(* IEC 61131-3 sources: json/test, 18 files *)

(* ---- CompareArray.st ---- *)
NAMESPACE Simatic.Ax.Json
    FUNCTION CompareArray : BOOL
        VAR_INPUT
            first : ARRAY[*] OF CHAR;
            scnd : ARRAY[*] OF CHAR;
            count : INT;
        END_VAR
        VAR_TEMP
            i : DINT;
            sFirst : DINT;
            sScnd : DINT;
            eFirst : DINT;
            eScnd : DINT;
            res : BOOL;
            _count : DINT;
        END_VAR

        sFirst := LOWER_BOUND(first, 1);
        sScnd := LOWER_BOUND(scnd, 1);
        eFirst := UPPER_BOUND(first, 1);
        eScnd := UPPER_BOUND(scnd, 1);

        _count := count;

        IF ((eFirst - sFirst + 1) < count) THEN
            CompareArray := FALSE;
            RETURN;
        END_IF;
        IF ((eScnd - sScnd + 1) < count) THEN
            CompareArray := FALSE;
            RETURN;
        END_IF;

        IF _count > (eFirst - sFirst + 1) THEN
            _count := eFirst - sFirst + 1;
        END_IF;

        FOR i := 0 TO _count - 1 DO
            res := first[i + sFirst] = scnd[i + sScnd];
            IF (res = FALSE) THEN
                CompareArray := FALSE;
                RETURN;
            END_IF;
        END_FOR;
        CompareArray := TRUE;
    END_FUNCTION
END_NAMESPACE

(* ---- FindKeyInBuffer.st ---- *)
USING Simatic.Ax.Conversion;
USING AxUnit.Assert;
USING System.Strings;
using Simatic.Ax.Json;

NAMESPACE Deserializer

{TestFixture}
CLASS Test_FindKeyInBuffer
    VAR protected
        doc : JsonDocument;
        testString : STRING := 'works!';
        buffer : ARRAY[1..999] OF CHAR;
    END_VAR

    METHOD PUBLIC ConvertStringToCharArray
        VAR_INPUT
            inputstring: string;
        end_var
        VAR_TEMP
            stringLength : int;
            index : Int;
        end_var

        stringLength := LengthOf(inputstring);

        FOR Index := 1 TO stringlength DO
            buffer[index] := inputstring[index];
        END_FOR;

    END_METHOD

    {Test}
    METHOD PUBLIC Test_ConvertStringToCharArray
            THIS.ConvertStringToCharArray(testString);
            Equal('w', buffer[1]);
            Equal('o', buffer[2]);
            Equal('r', buffer[3]);
            Equal('k', buffer[4]);
            Equal('s', buffer[5]);
            Equal('!', buffer[6]);
    END_METHOD

END_CLASS

{Test}
FUNCTION GetACharInString
    VAR_TEMP
        e : STRING := 'hallo';
        c : CHAR;
    end_var
        c := e[1];
        Equal(c, 'h');
END_FUNCTION

END_NAMESPACE

(* ---- StringAssert.st ---- *)
USING AxUnit.ResultFunctions;
USING System.Strings;

NAMESPACE AxUnit.Assert
    FUNCTION PUBLIC Equal
        VAR_INPUT
            actual : String;
            expected: String;
            {CallerFilePath}
            file : WSTRING[1024];
            {CallerLineNumber}
            line : INT;
        END_VAR

        IF actual = expected THEN
            axunit_Succeed();
        ELSE
            axunit_Fail(Concat('Expected ', ', but found '), file, line);
        END_IF;

    END_FUNCTION
END_NAMESPACE

(* ---- test.st ---- *)
USING AxUnit.Assert;

NAMESPACE Simatic.Ax.Json
    FUNCTION test : Int
        VAR_INPUT

        END_VAR
        test := 3;
    END_FUNCTION

    {TestFixture}
    CLASS MyTestFixture
        {Test}
        METHOD PUBLIC function_returns_alwasy_4
            Equal(expected := 4, actual := test());
            ; // AxUnit.Assert.Equal(y, x)
        END_METHOD
    END_CLASS

END_NAMESPACE

(* ---- TestFindKeyInBuffer.st ---- *)
USING Simatic.Ax.Conversion;
USING AxUnit.Assert;
USING System.Strings;
using Simatic.Ax.Json;

NAMESPACE Deserializer

{TestFixture}
CLASS Test_FindKeyInBuffer
    VAR protected
        doc : JsonDocument;
        key: STRING := 'key';
        testString : STRING := 'works!';
        buffer : ARRAY[0..999] OF CHAR;
    END_VAR

    {Test}
    Method Public Test_FindAKeyPosition_in_JSON_OneEntry
        VAR
            JSON_Entry: STRING := '{"Key1": "Element1"}';

            len:DINT;
            keyStart : int;
            keyEnd : int;
            keysFound: int;
        END_VAR

        len:= Strings.ToArray(str := JSON_Entry, arr := doc.buffer);

        keysFound := doc.FindKey(keyStart, keyEnd);

        //index is 0 based, not 1 based!
        Equal(2, keyStart);
        Equal(5, keyEnd);
        Equal(keysFound, 1);
    END_Method

    {Test}
    Method Public Test_FindKeysPosition_in_JSON_2Entries
        VAR
            JSON_Entry: STRING := '{"Key1": "Element1","Key2": 1234}';

            len:DINT;
            keyStart : int;
            keyEnd : int;
            keysFound: int;
        END_VAR

        len:= Strings.ToArray(str := JSON_Entry, arr := doc.buffer);

        keysFound := doc.FindKey(keyStart, keyEnd);

        //index is 0 based, not 1 based!
        Equal(21, keyStart);
        Equal(24, keyEnd);
        Equal(keysFound, 2);
    END_Method

    {Test}
    Method Public Test_KeyIsInIndexSpan_FindsKey
        VAR
            len:DINT;
            keyStart : int := 0;
            keyEnd : int := 2;
            keyFound: BOOL;

            test: bool := true;
        END_VAR

        len:= Strings.ToArray(str := key, arr := doc.buffer);

        keyFound := doc.KeyIsInIndexSpan(REF(key), keyStart, keyEnd);
        Equal(TRUE, keyFound);

        key := 'not';
        keyFound := doc.KeyIsInIndexSpan(REF(key), keyStart, keyEnd);
        Equal(FALSE, keyFound);
    END_Method

    //start with FindKey, in a string, Get Back Key and value. Make TryParse out of it (provide key). Nachteil: json wird jedes mal durchsucht. Test: Stringlänge! (Refto string?)

END_CLASS

{Test}
FUNCTION GetACharInString
    VAR_TEMP
        e : STRING := 'hallo';
        c : CHAR;
    end_var
        c := e[1];
        Equal(c, 'h');
END_FUNCTION

END_NAMESPACE

(* ---- Example.st ---- *)
USING Simatic.Ax.Json;
USING AxUnit.Assert;

NAMESPACE Simatic.Ax
    CLASS JsonExample
        VAR PUBLIC

        END_VAR
        VAR PROTECTED
            doc : JsonDocument;
            e1 : JsonDInt := (Key := 'Element1', Value := 1);
            e2 : JsonDInt := (Key := 'Element2', Value := 2);
            e3 : JsonDInt := (Key := 'Element3', Value := 3);
            o1 : JsonObject := (Key := 'NestedObject');

        END_VAR

        METHOD PUBLIC Init;
            // Example String:
            // {"Element1": 1, {"Element2": 2, "Element3": 3}}
            doc.AddElement(e1);
            doc.AddElement(o1);
            o1.AddElement(e2);
            o1.AddElement(e3);
        END_METHOD

        METHOD PUBLIC ToString : STRING
            ToString := doc.ToString();
        END_METHOD
    END_CLASS
END_NAMESPACE

NAMESPACE Simatic.Ax
    {TestFixture}
    CLASS TestExample
        VAR PROTECTED
            _ex : JsonExample;
        END_VAR

        {Test}
        METHOD PUBLIC TestExample_and_check_returned_string
            VAR_TEMP
                _expStr : STRING;
                _actStr : STRING;
            END_VAR
            _ex.Init();
            _expStr := '{"Element1": 1, "NestedObject": {"Element2": 2, "Element3": 3}}';
            _actStr := _ex.ToString();
            Equal(expected := _actStr, actual := _expStr);
        END_METHOD
    END_CLASS

END_NAMESPACE

(* ---- ItemTest.st ---- *)
USING AxUnit.Assert;
USING System.Strings;

NAMESPACE Simatic.Ax.Json
    {TestFixture}
    CLASS TestJsonElementsDint

        VAR PROTECTED
            e : Properties.DoubleInt := (value := 999, key := 'test');
        END_VAR

        {Test}
        METHOD PUBLIC Test_Tostring_with_999_expect_test_999
            Equal(expected := e.ToString(), actual := '"test": "999"');
        END_METHOD

        {Test}
        METHOD PUBLIC Test_Tostring_with_Minus_999_expect_test_Minus_999
            Equal(expected := e.ToString(), actual := '"test": "999"');
        END_METHOD

    END_CLASS
END_NAMESPACE

(* ---- ItemTestDint.st ---- *)
USING AxUnit.Assert;
USING System.Strings;

NAMESPACE Simatic.Ax.Json
    {TestFixture}
    CLASS TestJsonElementsDint

        VAR PROTECTED
            e : JsonDoubleInt := (value := 999, key := 'test');
            e2 : JsonDoubleInt := (value := -999, key := 'second_key');
        END_VAR

        {Test}
        METHOD PUBLIC Test_Tostring_with_999_expect_test_999
            VAR_TEMP
                _str : STRING;
            END_VAR
            _str := e.ToString();
            Equal(expected := _str, actual := '"test": 999');
        END_METHOD

        {Test}
        METHOD PUBLIC Test_Tostring_with_Minus_999_expect_test_Minus_999
            Equal(expected := e2.ToString(), actual := '"second_key": -999');
        END_METHOD

    END_CLASS
END_NAMESPACE

(* ---- ItemTestInt.st ---- *)
USING AxUnit.Assert;
USING System.Strings;
USING Simatic.Ax.Conversion;

NAMESPACE Simatic.Ax.Json
    {TestFixture}
    CLASS TestJsonElementsInt

        VAR PROTECTED
            e : JsonInt := (value := 999, key := 'test');
            e2 : JsonInt := (value := -999, key := 'second_key');
            s_test_999 : STRING := '"test": 999';
            s_test_minus_999 : STRING := '"second_key": -999';
            cmpBuff : ARRAY[0..20] OF CHAR;
            doc : JsonDocument;
        END_VAR

        {Test}
        METHOD PUBLIC Test_Tostring_with_999_expect_test_999
            VAR_TEMP
                _str : STRING;
            END_VAR
            _str := e.ToString();
            Equal(expected := _str, actual := s_test_999);
        END_METHOD

        {Test}
        METHOD PUBLIC Test_Tostring_with_Minus_999_expect_test_Minus_999
            Equal(expected := e2.ToString(), actual := s_test_minus_999);
        END_METHOD

        {Test}
        METHOD PUBLIC TestSerialize_s_test_999
            VAR_TEMP
                len : DINT;
                res : BOOL;
            END_VAR
            e.Serialize(REF(doc));

            len := Strings.ToArray(str := s_test_999, arr := cmpBuff);
            res := CompareArray(first := doc.buffer, scnd := cmpBuff, count := TO_INT(len));
            Equal(expected := TRUE, actual := res);

        END_METHOD

        {Test}
        METHOD PUBLIC TestSerialize_s_test_minus_999
            VAR_TEMP
                len : DINT;
                res : BOOL;
            END_VAR

            e2.Serialize(REF(doc));
            len := Strings.ToArray(str := s_test_minus_999, arr := cmpBuff);
            res := CompareArray(first := doc.buffer, scnd := cmpBuff, count := TO_INT(len));
            Equal(expected := TRUE, actual := res);

        END_METHOD
    END_CLASS
END_NAMESPACE

(* ---- ItemTestLint.st ---- *)
USING AxUnit.Assert;
USING System.Strings;

NAMESPACE Simatic.Ax.Json
    {TestFixture}
    CLASS TestJsonElementsLint

        VAR PROTECTED
            e : JsonLInt := (Value := 999, Key := 'test');
            e2 : JsonLInt := (Value := -999, Key := 'second_key');
        END_VAR

        {Test}
        METHOD PUBLIC Test_Tostring_with_999_expect_test_999
            VAR_TEMP
                _str : STRING;
            END_VAR
            _str := e.ToString();
            Equal(expected := _str, actual := '"test": 999');
        END_METHOD

        {Test}
        METHOD PUBLIC Test_Tostring_with_Minus_999_expect_test_Minus_999
            Equal(expected := e2.ToString(), actual := '"second_key": -999');
        END_METHOD

    END_CLASS
END_NAMESPACE

(* ---- ItemTestSint.st ---- *)
USING AxUnit.Assert;
USING System.Strings;
USING Simatic.Ax.Conversion;

NAMESPACE Simatic.Ax.Json
    {TestFixture}
    CLASS TestJsonElementsSInt

        VAR PROTECTED
            e : JsonSInt := (Value := SINT#127, Key := 'test');
            e2 : JsonSInt := (Value := SINT#-128, Key := 'second_key');
            s_test_127 : STRING := '"test": 127';
            s_test_minus_128 : STRING := '"second_key": -128';
            cmpBuff : ARRAY[0..20] OF CHAR;
            doc : JsonDocument;
        END_VAR

        {Test}
        METHOD PUBLIC Test_Tostring_with_999_expect_test_999
            VAR_TEMP
                _str : STRING;
            END_VAR
            _str := e.ToString();
            Equal(expected := _str, actual := s_test_127);
        END_METHOD

        {Test}
        METHOD PUBLIC Test_Tostring_with_Minus_999_expect_test_Minus_999
            Equal(expected := e2.ToString(), actual := s_test_minus_128);
        END_METHOD

        {Test}
        METHOD PUBLIC TestSerialize_s_test_999
            VAR_TEMP
                len : DINT;
                res : BOOL;
            END_VAR
            e.Serialize(REF(doc));

            len := Strings.ToArray(str := s_test_127, arr := cmpBuff);
            res := CompareArray(first := doc.buffer, scnd := cmpBuff, count := TO_INT(len));
            Equal(expected := TRUE, actual := res);

        END_METHOD

        {Test}
        METHOD PUBLIC TestSerialize_s_test_minus_999
            VAR_TEMP
                len : DINT;
                res : BOOL;
            END_VAR

            e2.Serialize(REF(doc));
            len := Strings.ToArray(str := s_test_minus_128, arr := cmpBuff);
            res := CompareArray(first := doc.buffer, scnd := cmpBuff, count := TO_INT(len));
            Equal(expected := TRUE, actual := res);

        END_METHOD
    END_CLASS
END_NAMESPACE

(* ---- ItemTestUSint.st ---- *)
USING AxUnit.Assert;
USING System.Strings;
USING Simatic.Ax.Conversion;

NAMESPACE Simatic.Ax.Json
    {TestFixture}
    CLASS TestJsonElementsUSInt

        VAR PROTECTED
            e : JsonUSInt := (Value := USINT#255, Key := 'test');
            e2 : JsonUSInt := (Value := USINT#0, Key := 'second_key');
            s_test_max : STRING := '"test": 255';
            s_test_minus_min : STRING := '"second_key": 0';
            cmpBuff : ARRAY[0..20] OF CHAR;
            doc : JsonDocument;
        END_VAR

        {Test}
        METHOD PUBLIC Test_Tostring_with_999_expect_test_999
            VAR_TEMP
                _str : STRING;
            END_VAR
            _str := e.ToString();
            Equal(expected := _str, actual := s_test_max);
        END_METHOD

        {Test}
        METHOD PUBLIC Test_Tostring_with_Minus_999_expect_test_Minus_999
            Equal(expected := e2.ToString(), actual := s_test_minus_min);
        END_METHOD

        {Test}
        METHOD PUBLIC TestSerialize_s_test_999
            VAR_TEMP
                len : DINT;
                res : BOOL;
            END_VAR
            e.Serialize(REF(doc));

            len := Strings.ToArray(str := s_test_max, arr := cmpBuff);
            res := CompareArray(first := doc.buffer, scnd := cmpBuff, count := TO_INT(len));
            Equal(expected := TRUE, actual := res);

        END_METHOD

        {Test}
        METHOD PUBLIC TestSerialize_s_test_minus_999
            VAR_TEMP
                len : DINT;
                res : BOOL;
            END_VAR

            e2.Serialize(REF(doc));
            len := Strings.ToArray(str := s_test_minus_min, arr := cmpBuff);
            res := CompareArray(first := doc.buffer, scnd := cmpBuff, count := TO_INT(len));
            Equal(expected := TRUE, actual := res);

        END_METHOD
    END_CLASS
END_NAMESPACE

(* ---- TestCompareArray.st ---- *)
USING AxUnit.Assert;
USING System.Strings;

NAMESPACE Simatic.Ax.Json
    {TestFixture}
    CLASS TestCompareArrayOfChar
        VAR
            a0_4_abcde : ARRAY[0..4] OF CHAR := ['a', 'b', 'c', 'd', 'e'];
            a0_4_abcdf : ARRAY[0..4] OF CHAR := ['a', 'b', 'c', 'd', 'f'];
            a0_4_12345 : ARRAY[0..4] OF CHAR := ['1', '2', '3', '4', '5'];
            a2_6_abcde : ARRAY[2..6] OF CHAR := ['a', 'b', 'c', 'd', 'e'];
            a2_6_12345 : ARRAY[2..6] OF CHAR := ['1', '2', '3', '4', '5'];
            a0_2_abc : ARRAY[0..2] OF CHAR := ['a', 'b', 'c'];
        END_VAR

        {Test}
        METHOD PUBLIC Copare_same_ArrayWithLengt5_Expect_TRUE
            VAR_TEMP
                res : BOOL;
            END_VAR
            res := CompareArray(a0_4_abcde, a0_4_abcde, 5);
            Equal(expected := TRUE, actual := res);

            res := CompareArray(a2_6_abcde, a2_6_abcde, 5);
            Equal(expected := TRUE, actual := res);
        END_METHOD

        {Test}
        METHOD PUBLIC Copare_different_ArrayWithLengt5_Expect_FALSE
            VAR_TEMP
                res : BOOL;
            END_VAR
            res := CompareArray(a0_4_abcde, a2_6_12345, 5);
            Equal(expected := FALSE, actual := res);

            res := CompareArray(a2_6_abcde, a0_4_12345, 5);
            Equal(expected := FALSE, actual := res);

            res := CompareArray(a0_4_abcde, a0_4_abcdf, 5);
            Equal(expected := FALSE, actual := res);

        END_METHOD

        {Test}
        METHOD PUBLIC Copare_different_ArrayWithLengt4_Expect_TRUE
            VAR_TEMP
                res : BOOL;
            END_VAR

            res := CompareArray(a0_4_abcde, a0_4_abcdf, 4);
            Equal(expected := TRUE, actual := res);

        END_METHOD

        {Test}
        METHOD PUBLIC Copare_same_ArrayWithLengt4_Expect_TRUE
            VAR_TEMP
                res : BOOL;
            END_VAR
            res := CompareArray(a0_4_abcde, a0_4_abcde, 4);
            Equal(expected := TRUE, actual := res);

            res := CompareArray(a2_6_abcde, a2_6_abcde, 4);
            Equal(expected := TRUE, actual := res);
        END_METHOD

        {Test}
        METHOD PUBLIC Copare_mixed_indices_ArrayWithLengt5_Expect_TRUE
            VAR_TEMP
                res : BOOL;
            END_VAR
            res := CompareArray(a0_4_abcde, a2_6_abcde, 5);
            Equal(expected := TRUE, actual := res);
        END_METHOD

        {Test}
        METHOD PUBLIC Copare_different_ArrayWithLengt4_Expect_FALSE
            VAR_TEMP
                res : BOOL;
            END_VAR
            res := CompareArray(a0_4_abcde, a2_6_12345, 4);
            Equal(expected := FALSE, actual := res);

            res := CompareArray(a2_6_abcde, a0_4_12345, 4);
            Equal(expected := FALSE, actual := res);
        END_METHOD

        {Test}
        METHOD PUBLIC Copare_different_lenght_ArrayWithLengt5_and_3_Expect_TRUE
            VAR_TEMP
                res : BOOL;
            END_VAR
            res := CompareArray(a0_4_abcde, a0_2_abc, 2);
            Equal(expected := TRUE, actual := res);

            res := CompareArray(a0_2_abc, a0_4_abcde, 2);
            Equal(expected := TRUE, actual := res);

            res := CompareArray(a0_4_abcde, a0_2_abc, 3);
            Equal(expected := TRUE, actual := res);

            res := CompareArray(a0_2_abc, a0_4_abcde, 3);
            Equal(expected := TRUE, actual := res);

            res := CompareArray(a0_4_abcde, a0_2_abc, 4);
            Equal(expected := FALSE, actual := res);

            res := CompareArray(a0_2_abc, a0_4_abcde, 4);
            Equal(expected := FALSE, actual := res);

            res := CompareArray(a0_4_abcde, a0_2_abc, 5);
            Equal(expected := FALSE, actual := res);

            res := CompareArray(a0_2_abc, a0_4_abcde, 5);
            Equal(expected := FALSE, actual := res);

            res := CompareArray(a0_4_abcde, a0_2_abc, 6);
            Equal(expected := FALSE, actual := res);

            res := CompareArray(a0_2_abc, a0_4_abcde, 6);
            Equal(expected := FALSE, actual := res);

        END_METHOD

    END_CLASS
END_NAMESPACE

(* ---- TestDoubleNestetdObject.st ---- *)
USING AxUnit.Assert;
USING System.Strings;
USING Simatic.Ax.Conversion;

NAMESPACE Simatic.Ax.Json
    {TestFixture}
    CLASS TestDoubleNestetdObject

        VAR PROTECTED
            e1 : JsonDInt := (Value := 999, Key := 'e1');
            o1 : JsonObject := (Key := 'O1');
            o2 : JsonObject := (Key := 'O2');
            o3 : JsonObject := (Key := 'O3');

            // {"O1": {"O2": "O3""e1" :}}
                                // 01234567890123456789012345678901234567890
            expString : STRING := '{"O1": {"O2": {"O3": {"e1": 999}}}}';

            actString : STRING;
            res : BOOL;
            doc : JsonDocument;
            cmpBuff : ARRAY[0..399] OF CHAR;
            len : DINT;
        END_VAR

        {Test}
        METHOD PUBLIC Test_Build_nested_object_And_expect_correct_JSON
            VAR_TEMP
                _to : IJsonElementMuteable;
                _elem : IJsonElement;
            END_VAR

            o3.AddElement(e1);
            o2.AddElement(o3);
            o1.AddElement(o2);
            doc.AddElement(o1);
            doc.Serialize(doc.buffer);

            len := Strings.ToArray(str := expString, arr := cmpBuff);
            res := CompareArray(first := doc.buffer, scnd := cmpBuff, count := TO_INT(len));
            Equal(expected := TRUE, actual := res);
        END_METHOD

    END_CLASS
END_NAMESPACE

(* ---- TestFindValueInBuffer.st ---- *)
USING Simatic.Ax.Conversion;
USING AxUnit.Assert;
USING System.Strings;
using Simatic.Ax.Json;

NAMESPACE Deserializer

{TestFixture}
CLASS Test_FindValueInBuffer
    VAR protected
        doc : JsonDocument;

        key: STRING;
        value: STRING;
        testIndex1: INT;
        testIndex2: INT;
    END_VAR

    {Test}
    Method Public Test_GetValueFromIndex_GetValue
        VAR
            len: DINT;
        END_VAR

        len:= Strings.ToArray(str := '1234', arr := doc.buffer);

        testIndex1:= 0; testIndex2 := 3;
        value:= doc.GetValueFromIndex(REF(testIndex1), REF(testIndex2));

        Equal('1234', value);

    END_Method

    {Test}
    Method Public Test_GetValueFromIndex_GetValue_withSpaces
        VAR
            len: DINT;
        END_VAR

        len:= Strings.ToArray(str := '    1234    ', arr := doc.buffer);

        testIndex1:= 0; testIndex2 := 10;
        value:= doc.GetValueFromIndex(REF(testIndex1), REF(testIndex2));

        Equal('1234', value);

    END_Method

    {Test}
    Method Public Test_GetValueFromIndex_GetValue_withQuotationMarks
        VAR
            len: DINT;
        END_VAR

        len:= Strings.ToArray(str := ' "1234"      ', arr := doc.buffer);

        testIndex1:= 0; testIndex2 := 10;
        value:= doc.GetValueFromIndex(REF(testIndex1), REF(testIndex2));

        Equal('1234', value);

    END_Method

END_CLASS

END_NAMESPACE

(* ---- TestJsonDocument.st ---- *)
USING AxUnit.Assert;
USING System.Strings;
USING Simatic.Ax.Conversion;

NAMESPACE Simatic.Ax.Json
    {TestFixture}
    CLASS TestJsonDocument

        VAR PROTECTED
            e : JsonDoubleInt := (value := 999, key := 'test');
            e2 : JsonDoubleInt := (value := -999, key := 'second_key');
            e3 : JsonDoubleInt := (value := 1, key := '3rd');
            doc : JsonDocument;
            o2 : JsonObject := (key := 'Name');

            iElem : IJsonElement;
            rElem : REF_TO JsonDoubleInt;
            expArray : ARRAY[0..399] OF CHAR;
            expArrayCnt : DINT;
            expString : STRING;
            actString : STRING;
            result : BOOL;

        END_VAR

        {Test}
        METHOD PUBLIC Test_Empty_object_ToString_Expect_empty_object

            // expected string
            expString := '{}';

            actString :=  doc.ToString();
            Equal(expected := expString, actual := actString);

            // Test Serialize
            expArrayCnt := Strings.ToArray(str := expString, arr := expArray);
            doc.Serialize(doc.buffer);
            result := CompareArray(first := doc.buffer, scnd := expArray, count := TO_INT(expArrayCnt));
            Equal(expected := TRUE, actual := result);

        END_METHOD

        {Test}
        METHOD PUBLIC Test_object_with_one_element_ToString_Expect_correct_string
            // expected string
            expString := '{"test": 999}';

            doc.AddElement(e);
            actString := doc.ToString();
            Equal(expected := expString, actual := actString);

            // Test Serialize
            expArrayCnt := Strings.ToArray(str := expString, arr := expArray);
            doc.Serialize(doc.buffer);
            result := CompareArray(first := doc.buffer, scnd := expArray, count := TO_INT(expArrayCnt));
            Equal(expected := TRUE, actual := result);
        END_METHOD

        {Test}
        METHOD PUBLIC Test_object_in_object_expect_nested_object
            // expected string
            expString := '{{}}';

            doc.AddElement(o2);
            Equal(expected := doc.ToString(), actual := expString);

            // Test Serialize
            expArrayCnt := Strings.ToArray(str := expString, arr := expArray);
            doc.Serialize(doc.buffer);
            result := CompareArray(first := doc.buffer, scnd := expArray, count := TO_INT(expArrayCnt));
            Equal(expected := TRUE, actual := result);
        END_METHOD

        {Test}
        METHOD PUBLIC Test_object_in_object_with_property_expect_nested_object
            // expected string
            expString := '{"Name": {"test": 999}}';

            doc.AddElement(o2);
            o2.AddElement(e);

            actString := doc.ToString();
            Equal(expected := actString, actual := expString);

            // Test Serialize
            expArrayCnt := Strings.ToArray(str := expString, arr := expArray);
            doc.Serialize(doc.buffer);
            result := CompareArray(first := doc.buffer, scnd := expArray, count := TO_INT(expArrayCnt));
            Equal(expected := TRUE, actual := result);
        END_METHOD

        {Test}
        METHOD PUBLIC Test_object_with_two_property_expect_object
            // expected string
            expString := '{"test": 999, "second_key": -999}';

            doc.AddElement(e);
            doc.AddElement(e2);
            Equal(expected := doc.ToString(), actual := expString);

            // Test Serialize
            expArrayCnt := Strings.ToArray(str := expString, arr := expArray);
            doc.Serialize(doc.buffer);
            result := CompareArray(first := doc.buffer, scnd := expArray, count := TO_INT(expArrayCnt));
            Equal(expected := TRUE, actual := result);
        END_METHOD

        {Test}
        METHOD PUBLIC Test_object_with_three_property_expect_object
            // expected string
            expString := '{"test": 999, "second_key": -999, "3rd": 1}';

            doc.AddElement(e);
            doc.AddElement(e2);
            doc.AddElement(e3);
            Equal(expected := doc.ToString(), actual := expString);

            // Test Serialize
            expArrayCnt := Strings.ToArray(str := expString, arr := expArray);
            doc.Serialize(doc.buffer);
            result := CompareArray(first := doc.buffer, scnd := expArray, count := TO_INT(expArrayCnt));
            Equal(expected := TRUE, actual := result);
        END_METHOD

        {Test}
        METHOD PUBLIC CreateTwoObjects_and_expect_correct_values
            // expected string
            expString := '{"test": 999, "second_key": -999}';

            doc.AddElement(e);
            doc.AddElement(e2);
            Equal(expected := doc.ToString(), actual := expString);

            // expected string
            expString := '"NestedObject": {"3rd": 1}';

            o2.key := 'NestedObject';
            o2.AddElement(e3);
            actString := o2.ToString();
            Equal(expected := expString, actual := actString);

            //            0        1         2         3         4         5         6         7
            //            1234567890123456789012345678901234567890123456789012345678901234567890
            expString := '{"test": 999, "second_key": -999, "NestedObject": {"3rd": 1}}';

            doc.AddElement(o2);
            actString := o2.ToString();

            actString := doc.ToString();
            Equal(expected := expString , actual := actString);

            // // Test Serialize
            // expArrayCnt := Strings.ToArray(str := expString, arr := expArray);
            // doc.Serialize(doc.buffer);
            // result := CompareArray(first := doc.buffer, scnd := expArray, count := TO_INT(expArrayCnt));
            // Equal(expected := TRUE, actual := result);
        END_METHOD
    END_CLASS
END_NAMESPACE

(* ---- TestJsonLongDocument.st ---- *)
USING AxUnit.Assert;
USING System.Strings;
USING Simatic.Ax.Conversion;
NAMESPACE Simatic.Ax.Json
    {TestFixture}
    CLASS TestJsonLongDocument

        VAR PROTECTED
            e1 : JsonInt := (Key := 'elem1', Value := 0);
            e2 : JsonLInt := (Key := 'elem2', Value := 1);
            e3 : JsonDInt := (Key := 'elem3', Value := 2);
            doc :JsonDocument;
        END_VAR

        METHOD PUBLIC MyMethod
            doc.AddElement(e1);
            doc.AddElement(e2);
            doc.AddElement(e3);
            doc.Serialize(doc.buffer); //--> {elem1: 0, elem2: 1, elem3: 2}\n
            // nice to have --> doc.Deserialize('{elem1: 99, elem2: 100, elem3: 111}\n')
        END_METHOD

    END_CLASS

END_NAMESPACE

(* ---- TestJsonObject.st ---- *)
USING AxUnit.Assert;
USING System.Strings;
USING Simatic.Ax.Conversion;

NAMESPACE Simatic.Ax.Json
    {TestFixture}
    CLASS TestJsonObject

        VAR PROTECTED
            e : JsonDoubleInt := (value := 999, key := 'test');
            e2 : JsonDoubleInt := (value := -999, key := 'second_key');
            e3 : JsonDoubleInt := (value := 1, key := '3rd');
            o : JsonObject := (key := 'Name');
            doc : JsonDocument;
            cmpBuff : ARRAY[0..399] OF CHAR;
            len : DINT;
        END_VAR

        {Test}
        METHOD PUBLIC Test_Empty_object_ToString_Expect_empty_object
            VAR_TEMP
                _expStr : STRING;
                _actStr : STRING;
            END_VAR

            // {}
            _expStr := '{}';
            _actStr := o.ToString();
            Equal(expected := _actStr, actual := _expStr);
        END_METHOD

        {Test}
        METHOD PUBLIC Test_Object_with_one_element
            VAR_TEMP
                _expStr : STRING;
                _actStr : STRING;
            END_VAR
            o.AddElement(e);
            _expStr := '"Name": {"test": 999}';
            _actStr := o.ToString();
            Equal(expected := _actStr, actual := _expStr);
        END_METHOD

        {Test}
        METHOD PUBLIC Test_Object_with_three_elements
            VAR_TEMP
                _expStr : STRING;
                _actStr : STRING;
                _i, _j : INT;
            END_VAR
            o.AddElement(e);
            o.AddElement(e2);
            o.AddElement(e3);
            _expStr := '"Name": {"test": 999, "second_key": -999, "3rd": 1}';
            _expStr := StartOf(_expStr, 5);

            _i := LengthOf(_expStr);

            _actStr := StartOf(o.ToString(), LengthOf(_expStr));
            _j := LengthOf(_actStr);
            Equal(expected := _actStr, actual := _expStr);
        END_METHOD

        {Test}
        METHOD PUBLIC Test_Serialize_Object_with_three_elements
            VAR_TEMP
                _expStr : STRING;
                _actStr : STRING;
                _i, _j : INT;
                _res : BOOL;
            END_VAR
            THIS.Test_Object_with_three_elements();
            _expStr := '"Name": {"test": 999, "second_key": -999, "3rd": 1}';

            o.Serialize(REF(doc));

            len := Strings.ToArray(str := _expStr, arr := cmpBuff);
            _res := CompareArray(first := doc.buffer, scnd := cmpBuff, count := TO_INT(len));
            Equal(expected := TRUE, actual := _res);
        END_METHOD

    END_CLASS
END_NAMESPACE
